//     Term 17 (APS4322-7000)/APS Outputs/Current D 0X1 <-> Data Pointer/DCurrentSetPoints[1]
//     Term 17 (APS4322-7000)/APS Outputs/Current D 0X2 <-> Data Pointer/DCurrentSetPoints[2]
//     Term 17 (APS4322-7000)/APS Outputs/Current D 1X0 <-> Data Pointer/DCurrentSetPoints[6]
//     Term 17 (APS4322-7000)/APS Outputs/Current D 1X1 <-> Data Pointer/DCurrentSetPoints[7]
//     Term 17 (APS4322-7000)/APS Outputs/Current D 1X2 <-> Data Pointer/DCurrentSetPoints[8]
//     Term 17 (APS4322-7000)/APS Outputs/Current D 2X0 <-> Data Pointer/DCurrentSetPoints[12]
//     Term 17 (APS4322-7000)/APS Outputs/Current D 2X1 <-> Data Pointer/DCurrentSetPoints[13]
//     Term 17 (APS4322-7000)/APS Outputs/Current D 2X2 <-> Data Pointer/DCurrentSetPoints[14]
//     Term 17 (APS4322-7000)/APS Outputs/Current D 3X0 <-> Data Pointer/DCurrentSetPoints[18]
//     Term 17 (APS4322-7000)/APS Outputs/Current D 3X1 <-> Data Pointer/DCurrentSetPoints[19]
//     Term 17 (APS4322-7000)/APS Outputs/Current D 3X2 <-> Data Pointer/DCurrentSetPoints[20]
//     Term 17 (APS4322-7000)/APS Outputs/Current D 0Y0 <-> Data Pointer/DCurrentSetPoints[3]
//     Term 17 (APS4322-7000)/APS Outputs/Current D 0Y1 <-> Data Pointer/DCurrentSetPoints[4]
//     Term 17 (APS4322-7000)/APS Outputs/Current D 0Y2 <-> Data Pointer/DCurrentSetPoints[5]
//     Term 17 (APS4322-7000)/APS Outputs/Current D 1Y0 <-> Data Pointer/DCurrentSetPoints[9]
//     Term 17 (APS4322-7000)/APS Outputs/Current D 1Y1 <-> Data Pointer/DCurrentSetPoints[10]
//     Term 17 (APS4322-7000)/APS Outputs/Current D 1Y2 <-> Data Pointer/DCurrentSetPoints[11]
//     Term 17 (APS4322-7000)/APS Outputs/Current D 2Y0 <-> Data Pointer/DCurrentSetPoints[15]
//     Term 17 (APS4322-7000)/APS Outputs/Current D 2Y1 <-> Data Pointer/DCurrentSetPoints[16]
//     Term 17 (APS4322-7000)/APS Outputs/Current D 2Y2 <-> Data Pointer/DCurrentSetPoints[17]
//     Term 17 (APS4322-7000)/APS Outputs/Current D 3Y0 <-> Data Pointer/DCurrentSetPoints[21]
//     Term 17 (APS4322-7000)/APS Outputs/Current D 3Y1 <-> Data Pointer/DCurrentSetPoints[22]
//     Term 17 (APS4322-7000)/APS Outputs/Current D 3Y2 <-> Data Pointer/DCurrentSetPoints[23]
//     Term 17 (APS4322-7000)/APS Outputs/Current Q 0X0 <-> Data Pointer/QCurrentSetPoints[0]
//     Term 17 (APS4322-7000)/APS Outputs/Current Q 0X1 <-> Data Pointer/QCurrentSetPoints[1]
//     Term 17 (APS4322-7000)/APS Outputs/Current Q 0X2 <-> Data Pointer/QCurrentSetPoints[2]
//     Term 17 (APS4322-7000)/APS Outputs/Current Q 1X0 <-> Data Pointer/QCurrentSetPoints[6]
//     Term 17 (APS4322-7000)/APS Outputs/Current Q 1X1 <-> Data Pointer/QCurrentSetPoints[7]
//     Term 17 (APS4322-7000)/APS Outputs/Current Q 1X2 <-> Data Pointer/QCurrentSetPoints[8]
//     Term 17 (APS4322-7000)/APS Outputs/Current Q 2X0 <-> Data Pointer/QCurrentSetPoints[12]
//     Term 17 (APS4322-7000)/APS Outputs/Current Q 2X1 <-> Data Pointer/QCurrentSetPoints[13]
//     Term 17 (APS4322-7000)/APS Outputs/Current Q 2X2 <-> Data Pointer/QCurrentSetPoints[14]
//     Term 17 (APS4322-7000)/APS Outputs/Current Q 3X0 <-> Data Pointer/QCurrentSetPoints[18]
//     Term 17 (APS4322-7000)/APS Outputs/Current Q 3X1 <-> Data Pointer/QCurrentSetPoints[19]
//     Term 17 (APS4322-7000)/APS Outputs/Current Q 3X2 <-> Data Pointer/QCurrentSetPoints[20]
//     Term 17 (APS4322-7000)/APS Outputs/Current Q 0Y0 <-> Data Pointer/QCurrentSetPoints[3]
//     Term 17 (APS4322-7000)/APS Outputs/Current Q 0Y1 <-> Data Pointer/QCurrentSetPoints[4]
//     Term 17 (APS4322-7000)/APS Outputs/Current Q 0Y2 <-> Data Pointer/QCurrentSetPoints[5]
//     Term 17 (APS4322-7000)/APS Outputs/Current Q 1Y0 <-> Data Pointer/QCurrentSetPoints[9]
//     Term 17 (APS4322-7000)/APS Outputs/Current Q 1Y1 <-> Data Pointer/QCurrentSetPoints[10]
//     Term 17 (APS4322-7000)/APS Outputs/Current Q 1Y2 <-> Data Pointer/QCurrentSetPoints[11]
//     Term 17 (APS4322-7000)/APS Outputs/Current Q 2Y0 <-> Data Pointer/QCurrentSetPoints[15]
//     Term 17 (APS4322-7000)/APS Outputs/Current Q 2Y1 <-> Data Pointer/QCurrentSetPoints[16]
//     Term 17 (APS4322-7000)/APS Outputs/Current Q 2Y2 <-> Data Pointer/QCurrentSetPoints[17]
//     Term 17 (APS4322-7000)/APS Outputs/Current Q 3Y0 <-> Data Pointer/QCurrentSetPoints[21]
//     Term 17 (APS4322-7000)/APS Outputs/Current Q 3Y1 <-> Data Pointer/QCurrentSetPoints[22]
//     Term 17 (APS4322-7000)/APS Outputs/Current Q 3Y2 <-> Data Pointer/QCurrentSetPoints[23]
//     Term 17 (APS4322-7000)/APS Outputs/PhiE 0X0 <-> Data Pointer/PhiSetPoints[0]
//     Term 17 (APS4322-7000)/APS Outputs/PhiE 0X1 <-> Data Pointer/PhiSetPoints[1]
//     Term 17 (APS4322-7000)/APS Outputs/PhiE 0X2 <-> Data Pointer/PhiSetPoints[2]
//     Term 17 (APS4322-7000)/APS Outputs/PhiE 1X0 <-> Data Pointer/PhiSetPoints[6]
//     Term 17 (APS4322-7000)/APS Outputs/PhiE 1X1 <-> Data Pointer/PhiSetPoints[7]
//     Term 17 (APS4322-7000)/APS Outputs/PhiE 1X2 <-> Data Pointer/PhiSetPoints[8]
//     Term 17 (APS4322-7000)/APS Outputs/PhiE 2X0 <-> Data Pointer/PhiSetPoints[12]
//     Term 17 (APS4322-7000)/APS Outputs/PhiE 2X1 <-> Data Pointer/PhiSetPoints[13]
//     Term 17 (APS4322-7000)/APS Outputs/PhiE 2X2 <-> Data Pointer/PhiSetPoints[14]
//     Term 17 (APS4322-7000)/APS Outputs/PhiE 3X0 <-> Data Pointer/PhiSetPoints[18]
//     Term 17 (APS4322-7000)/APS Outputs/PhiE 3X1 <-> Data Pointer/PhiSetPoints[19]
//     Term 17 (APS4322-7000)/APS Outputs/PhiE 3X2 <-> Data Pointer/PhiSetPoints[20]
//     Term 17 (APS4322-7000)/APS Outputs/PhiE 0Y0 <-> Data Pointer/PhiSetPoints[3]
//     Term 17 (APS4322-7000)/APS Outputs/PhiE 0Y1 <-> Data Pointer/PhiSetPoints[4]
//     Term 17 (APS4322-7000)/APS Outputs/PhiE 0Y2 <-> Data Pointer/PhiSetPoints[5]
//     Term 17 (APS4322-7000)/APS Outputs/PhiE 1Y0 <-> Data Pointer/PhiSetPoints[9]
//     Term 17 (APS4322-7000)/APS Outputs/PhiE 1Y1 <-> Data Pointer/PhiSetPoints[10]
//     Term 17 (APS4322-7000)/APS Outputs/PhiE 1Y2 <-> Data Pointer/PhiSetPoints[11]
//     Term 17 (APS4322-7000)/APS Outputs/PhiE 2Y0 <-> Data Pointer/PhiSetPoints[15]
//     Term 17 (APS4322-7000)/APS Outputs/PhiE 2Y1 <-> Data Pointer/PhiSetPoints[16]
//     Term 17 (APS4322-7000)/APS Outputs/PhiE 2Y2 <-> Data Pointer/PhiSetPoints[17]
//     Term 17 (APS4322-7000)/APS Outputs/PhiE 3Y0 <-> Data Pointer/PhiSetPoints[21]
//     Term 17 (APS4322-7000)/APS Outputs/PhiE 3Y1 <-> Data Pointer/PhiSetPoints[22]
//     Term 17 (APS4322-7000)/APS Outputs/PhiE 3Y2 <-> Data Pointer/PhiSetPoints[23]
//     Term 17 (APS4322-7000)/Term 18 (APS4322-5000)/FB Inputs/A{0..8 step 2} X-Field <-> Data Pointer/HallSensorFieldsXYZ[{0..12 step 3}]  (5 links)
//     Term 17 (APS4322-7000)/Term 18 (APS4322-5000)/FB Inputs/A{0..8 step 2} Y-Field <-> Data Pointer/HallSensorFieldsXYZ[{1..13 step 3}]  (5 links)
//     Term 17 (APS4322-7000)/Term 18 (APS4322-5000)/FB Inputs/A{0..8 step 2} Z-Field <-> Data Pointer/HallSensorFieldsXYZ[{2..14 step 3}]  (5 links)
//     Term 17 (APS4322-7000)/Term 18 (APS4322-5000)/FB Inputs/B{1..9 step 2} X-Field <-> Data Pointer/HallSensorFieldsXYZ[{15..27 step 3}]  (5 links)
//     Term 17 (APS4322-7000)/Term 18 (APS4322-5000)/FB Inputs/B{1..9 step 2} Y-Field <-> Data Pointer/HallSensorFieldsXYZ[{16..28 step 3}]  (5 links)
//     Term 17 (APS4322-7000)/Term 18 (APS4322-5000)/FB Inputs/B{1..9 step 2} Z-Field <-> Data Pointer/HallSensorFieldsXYZ[{17..29 step 3}]  (5 links)
//     Term 17 (APS4322-7000)/Term 18 (APS4322-5000)/FB Inputs/C{0..8 step 2} X-Field <-> Data Pointer/HallSensorFieldsXYZ[{30..42 step 3}]  (5 links)
//     Term 17 (APS4322-7000)/Term 18 (APS4322-5000)/FB Inputs/C{0..8 step 2} Y-Field <-> Data Pointer/HallSensorFieldsXYZ[{31..43 step 3}]  (5 links)
//     Term 17 (APS4322-7000)/Term 18 (APS4322-5000)/FB Inputs/C{0..8 step 2} Z-Field <-> Data Pointer/HallSensorFieldsXYZ[{32..44 step 3}]  (5 links)
//     Term 17 (APS4322-7000)/Term 18 (APS4322-5000)/FB Inputs/D{1..9 step 2} X-Field <-> Data Pointer/HallSensorFieldsXYZ[{45..57 step 3}]  (5 links)
//     Term 17 (APS4322-7000)/Term 18 (APS4322-5000)/FB Inputs/D{1..9 step 2} Y-Field <-> Data Pointer/HallSensorFieldsXYZ[{46..58 step 3}]  (5 links)
//     Term 17 (APS4322-7000)/Term 18 (APS4322-5000)/FB Inputs/D{1..9 step 2} Z-Field <-> Data Pointer/HallSensorFieldsXYZ[{47..59 step 3}]  (5 links)
//     Term 17 (APS4322-7000)/Term 18 (APS4322-5000)/FB Inputs/E{0..8 step 2} X-Field <-> Data Pointer/HallSensorFieldsXYZ[{60..72 step 3}]  (5 links)
//     Term 17 (APS4322-7000)/Term 18 (APS4322-5000)/FB Inputs/E{0..8 step 2} Y-Field <-> Data Pointer/HallSensorFieldsXYZ[{61..73 step 3}]  (5 links)
//     Term 17 (APS4322-7000)/Term 18 (APS4322-5000)/FB Inputs/E{0..8 step 2} Z-Field <-> Data Pointer/HallSensorFieldsXYZ[{62..74 step 3}]  (5 links)
//     Term 17 (APS4322-7000)/Term 18 (APS4322-5000)/FB Inputs/F{1..9 step 2} X-Field <-> Data Pointer/HallSensorFieldsXYZ[{75..87 step 3}]  (5 links)
//     Term 17 (APS4322-7000)/Term 18 (APS4322-5000)/FB Inputs/F{1..9 step 2} Y-Field <-> Data Pointer/HallSensorFieldsXYZ[{76..88 step 3}]  (5 links)
//     Term 17 (APS4322-7000)/Term 18 (APS4322-5000)/FB Inputs/F{1..9 step 2} Z-Field <-> Data Pointer/HallSensorFieldsXYZ[{77..89 step 3}]  (5 links)
//     Term 17 (APS4322-7000)/Term 18 (APS4322-5000)/FB Inputs/G{0..8 step 2} X-Field <-> Data Pointer/HallSensorFieldsXYZ[{90..102 step 3}]  (5 links)
//     Term 17 (APS4322-7000)/Term 18 (APS4322-5000)/FB Inputs/G{0..8 step 2} Y-Field <-> Data Pointer/HallSensorFieldsXYZ[{91..103 step 3}]  (5 links)
//     Term 17 (APS4322-7000)/Term 18 (APS4322-5000)/FB Inputs/G{0..8 step 2} Z-Field <-> Data Pointer/HallSensorFieldsXYZ[{92..104 step 3}]  (5 links)
//     Term 17 (APS4322-7000)/Term 18 (APS4322-5000)/FB Inputs/H{1..9 step 2} X-Field <-> Data Pointer/HallSensorFieldsXYZ[{105..117 step 3}]  (5 links)
//     Term 17 (APS4322-7000)/Term 18 (APS4322-5000)/FB Inputs/H{1..9 step 2} Y-Field <-> Data Pointer/HallSensorFieldsXYZ[{106..118 step 3}]  (5 links)
//     Term 17 (APS4322-7000)/Term 18 (APS4322-5000)/FB Inputs/H{1..9 step 2} Z-Field <-> Data Pointer/HallSensorFieldsXYZ[{107..119 step 3}]  (5 links)
//     Term 17 (APS4322-7000)/Term 18 (APS4322-5000)/FB Inputs/I{0..8 step 2} X-Field <-> Data Pointer/HallSensorFieldsXYZ[{120..132 step 3}]  (5 links)
//     Term 17 (APS4322-7000)/Term 18 (APS4322-5000)/FB Inputs/I{0..8 step 2} Y-Field <-> Data Pointer/HallSensorFieldsXYZ[{121..133 step 3}]  (5 links)
//     Term 17 (APS4322-7000)/Term 18 (APS4322-5000)/FB Inputs/I{0..8 step 2} Z-Field <-> Data Pointer/HallSensorFieldsXYZ[{122..134 step 3}]  (5 links)
//     Term 17 (APS4322-7000)/Term 18 (APS4322-5000)/FB Inputs/J{1..9 step 2} X-Field <-> Data Pointer/HallSensorFieldsXYZ[{135..147 step 3}]  (5 links)
//     Term 17 (APS4322-7000)/Term 18 (APS4322-5000)/FB Inputs/J{1..9 step 2} Y-Field <-> Data Pointer/HallSensorFieldsXYZ[{136..148 step 3}]  (5 links)
//     Term 17 (APS4322-7000)/Term 18 (APS4322-5000)/FB Inputs/J{1..9 step 2} Z-Field <-> Data Pointer/HallSensorFieldsXYZ[{137..149 step 3}]  (5 links)
//     Term 17 (APS4322-7000)/Term 18 (APS4322-5000)/FB Inputs/Status <-> Data Pointer/FeedbackStatus
//   Device 2 (EtherCAT) <-> TcCOM Objects/XPlanar/Part1/Tile4
//     Term 19 (APS4322-7000)/APS Comm Inputs/CommStatusWord <-> Data Pointer/MoverCommStatusWord
//     Term 19 (APS4322-7000)/APS Comm Inputs/Data {1..4} <-> Data Pointer/MoverCommDataIn[{0..3}]  (4 links)
//     Term 19 (APS4322-7000)/APS Comm Outputs/CommControlWord <-> Data Pointer/MoverCommControlWord
//     Term 19 (APS4322-7000)/APS Comm Outputs/Data 1 <-> Data Pointer/MoverCommDataOut
//     Term 19 (APS4322-7000)/APS Diagdata/DC Link Voltage <-> Data Pointer/DcLinkVoltage
//     Term 19 (APS4322-7000)/APS Diagdata/Power supply current <-> Data Pointer/PowerSupplyCurrent
//     Term 19 (APS4322-7000)/APS Inputs/StatusWord <-> Data Pointer/PowerUnitStatusWord
//     Term 19 (APS4322-7000)/APS Outputs/ControlWord <-> Data Pointer/PowerUnitControlWord
//     Term 19 (APS4322-7000)/APS Outputs/Current D 0X0 <-> Data Pointer/DCurrentSetPoints[0]
//     Term 19 (APS4322-7000)/APS Outputs/Current D 0X1 <-> Data Pointer/DCurrentSetPoints[1]
//     Term 19 (APS4322-7000)/APS Outputs/Current D 0X2 <-> Data Pointer/DCurrentSetPoints[2]
//     Term 19 (APS4322-7000)/APS Outputs/Current D 1X0 <-> Data Pointer/DCurrentSetPoints[6]
//     Term 19 (APS4322-7000)/APS Outputs/Current D 1X1 <-> Data Pointer/DCurrentSetPoints[7]
//     Term 19 (APS4322-7000)/APS Outputs/Current D 1X2 <-> Data Pointer/DCurrentSetPoints[8]
//     Term 19 (APS4322-7000)/APS Outputs/Current D 2X0 <-> Data Pointer/DCurrentSetPoints[12]
//     Term 19 (APS4322-7000)/APS Outputs/Current D 2X1 <-> Data Pointer/DCurrentSetPoints[13]
//     Term 19 (APS4322-7000)/APS Outputs/Current D 2X2 <-> Data Pointer/DCurrentSetPoints[14]
//     Term 19 (APS4322-7000)/APS Outputs/Current D 3X0 <-> Data Pointer/DCurrentSetPoints[18]
//     Term 19 (APS4322-7000)/APS Outputs/Current D 3X1 <-> Data Pointer/DCurrentSetPoints[19]
//     Term 19 (APS4322-7000)/APS Outputs/Current D 3X2 <-> Data Pointer/DCurrentSetPoints[20]
//     Term 19 (APS4322-7000)/APS Outputs/Current D 0Y0 <-> Data Pointer/DCurrentSetPoints[3]
//     Term 19 (APS4322-7000)/APS Outputs/Current D 0Y1 <-> Data Pointer/DCurrentSetPoints[4]
//     Term 19 (APS4322-7000)/APS Outputs/Current D 0Y2 <-> Data Pointer/DCurrentSetPoints[5]
//     Term 19 (APS4322-7000)/APS Outputs/Current D 1Y0 <-> Data Pointer/DCurrentSetPoints[9]
//     Term 19 (APS4322-7000)/APS Outputs/Current D 1Y1 <-> Data Pointer/DCurrentSetPoints[10]
//     Term 19 (APS4322-7000)/APS Outputs/Current D 1Y2 <-> Data Pointer/DCurrentSetPoints[11]
//     Term 19 (APS4322-7000)/APS Outputs/Current D 2Y0 <-> Data Pointer/DCurrentSetPoints[15]
//     Term 19 (APS4322-7000)/APS Outputs/Current D 2Y1 <-> Data Pointer/DCurrentSetPoints[16]
//     Term 19 (APS4322-7000)/APS Outputs/Current D 2Y2 <-> Data Pointer/DCurrentSetPoints[17]
//     Term 19 (APS4322-7000)/APS Outputs/Current D 3Y0 <-> Data Pointer/DCurrentSetPoints[21]
//     Term 19 (APS4322-7000)/APS Outputs/Current D 3Y1 <-> Data Pointer/DCurrentSetPoints[22]
//     Term 19 (APS4322-7000)/APS Outputs/Current D 3Y2 <-> Data Pointer/DCurrentSetPoints[23]
//     Term 19 (APS4322-7000)/APS Outputs/Current Q 0X0 <-> Data Pointer/QCurrentSetPoints[0]
//     Term 19 (APS4322-7000)/APS Outputs/Current Q 0X1 <-> Data Pointer/QCurrentSetPoints[1]
//     Term 19 (APS4322-7000)/APS Outputs/Current Q 0X2 <-> Data Pointer/QCurrentSetPoints[2]
//     Term 19 (APS4322-7000)/APS Outputs/Current Q 1X0 <-> Data Pointer/QCurrentSetPoints[6]
//     Term 19 (APS4322-7000)/APS Outputs/Current Q 1X1 <-> Data Pointer/QCurrentSetPoints[7]
//     Term 19 (APS4322-7000)/APS Outputs/Current Q 1X2 <-> Data Pointer/QCurrentSetPoints[8]
//     Term 19 (APS4322-7000)/APS Outputs/Current Q 2X0 <-> Data Pointer/QCurrentSetPoints[12]
//     Term 19 (APS4322-7000)/APS Outputs/Current Q 2X1 <-> Data Pointer/QCurrentSetPoints[13]
//     Term 19 (APS4322-7000)/APS Outputs/Current Q 2X2 <-> Data Pointer/QCurrentSetPoints[14]
//     Term 19 (APS4322-7000)/APS Outputs/Current Q 3X0 <-> Data Pointer/QCurrentSetPoints[18]
//     Term 19 (APS4322-7000)/APS Outputs/Current Q 3X1 <-> Data Pointer/QCurrentSetPoints[19]
//     Term 19 (APS4322-7000)/APS Outputs/Current Q 3X2 <-> Data Pointer/QCurrentSetPoints[20]
//     Term 19 (APS4322-7000)/APS Outputs/Current Q 0Y0 <-> Data Pointer/QCurrentSetPoints[3]
//     Term 19 (APS4322-7000)/APS Outputs/Current Q 0Y1 <-> Data Pointer/QCurrentSetPoints[4]
//     Term 19 (APS4322-7000)/APS Outputs/Current Q 0Y2 <-> Data Pointer/QCurrentSetPoints[5]
//     Term 19 (APS4322-7000)/APS Outputs/Current Q 1Y0 <-> Data Pointer/QCurrentSetPoints[9]
//     Term 19 (APS4322-7000)/APS Outputs/Current Q 1Y1 <-> Data Pointer/QCurrentSetPoints[10]
//     Term 19 (APS4322-7000)/APS Outputs/Current Q 1Y2 <-> Data Pointer/QCurrentSetPoints[11]
//     Term 19 (APS4322-7000)/APS Outputs/Current Q 2Y0 <-> Data Pointer/QCurrentSetPoints[15]
//     Term 19 (APS4322-7000)/APS Outputs/Current Q 2Y1 <-> Data Pointer/QCurrentSetPoints[16]
//     Term 19 (APS4322-7000)/APS Outputs/Current Q 2Y2 <-> Data Pointer/QCurrentSetPoints[17]
//     Term 19 (APS4322-7000)/APS Outputs/Current Q 3Y0 <-> Data Pointer/QCurrentSetPoints[21]
//     Term 19 (APS4322-7000)/APS Outputs/Current Q 3Y1 <-> Data Pointer/QCurrentSetPoints[22]
//     Term 19 (APS4322-7000)/APS Outputs/Current Q 3Y2 <-> Data Pointer/QCurrentSetPoints[23]
//     Term 19 (APS4322-7000)/APS Outputs/PhiE 0X0 <-> Data Pointer/PhiSetPoints[0]
//     Term 19 (APS4322-7000)/APS Outputs/PhiE 0X1 <-> Data Pointer/PhiSetPoints[1]
//     Term 19 (APS4322-7000)/APS Outputs/PhiE 0X2 <-> Data Pointer/PhiSetPoints[2]
//     Term 19 (APS4322-7000)/APS Outputs/PhiE 1X0 <-> Data Pointer/PhiSetPoints[6]
//     Term 19 (APS4322-7000)/APS Outputs/PhiE 1X1 <-> Data Pointer/PhiSetPoints[7]
//     Term 19 (APS4322-7000)/APS Outputs/PhiE 1X2 <-> Data Pointer/PhiSetPoints[8]
//     Term 19 (APS4322-7000)/APS Outputs/PhiE 2X0 <-> Data Pointer/PhiSetPoints[12]
//     Term 19 (APS4322-7000)/APS Outputs/PhiE 2X1 <-> Data Pointer/PhiSetPoints[13]
//     Term 19 (APS4322-7000)/APS Outputs/PhiE 2X2 <-> Data Pointer/PhiSetPoints[14]
//     Term 19 (APS4322-7000)/APS Outputs/PhiE 3X0 <-> Data Pointer/PhiSetPoints[18]
//     Term 19 (APS4322-7000)/APS Outputs/PhiE 3X1 <-> Data Pointer/PhiSetPoints[19]
//     Term 19 (APS4322-7000)/APS Outputs/PhiE 3X2 <-> Data Pointer/PhiSetPoints[20]
//     Term 19 (APS4322-7000)/APS Outputs/PhiE 0Y0 <-> Data Pointer/PhiSetPoints[3]
//     Term 19 (APS4322-7000)/APS Outputs/PhiE 0Y1 <-> Data Pointer/PhiSetPoints[4]
//     Term 19 (APS4322-7000)/APS Outputs/PhiE 0Y2 <-> Data Pointer/PhiSetPoints[5]
//     Term 19 (APS4322-7000)/APS Outputs/PhiE 1Y0 <-> Data Pointer/PhiSetPoints[9]
//     Term 19 (APS4322-7000)/APS Outputs/PhiE 1Y1 <-> Data Pointer/PhiSetPoints[10]
//     Term 19 (APS4322-7000)/APS Outputs/PhiE 1Y2 <-> Data Pointer/PhiSetPoints[11]
//     Term 19 (APS4322-7000)/APS Outputs/PhiE 2Y0 <-> Data Pointer/PhiSetPoints[15]
//     Term 19 (APS4322-7000)/APS Outputs/PhiE 2Y1 <-> Data Pointer/PhiSetPoints[16]
//     Term 19 (APS4322-7000)/APS Outputs/PhiE 2Y2 <-> Data Pointer/PhiSetPoints[17]
//     Term 19 (APS4322-7000)/APS Outputs/PhiE 3Y0 <-> Data Pointer/PhiSetPoints[21]
//     Term 19 (APS4322-7000)/APS Outputs/PhiE 3Y1 <-> Data Pointer/PhiSetPoints[22]
//     Term 19 (APS4322-7000)/APS Outputs/PhiE 3Y2 <-> Data Pointer/PhiSetPoints[23]
//     Term 19 (APS4322-7000)/Term 20 (APS4322-5000)/FB Inputs/A{0..8 step 2} X-Field <-> Data Pointer/HallSensorFieldsXYZ[{0..12 step 3}]  (5 links)
//     Term 19 (APS4322-7000)/Term 20 (APS4322-5000)/FB Inputs/A{0..8 step 2} Y-Field <-> Data Pointer/HallSensorFieldsXYZ[{1..13 step 3}]  (5 links)
//     Term 19 (APS4322-7000)/Term 20 (APS4322-5000)/FB Inputs/A{0..8 step 2} Z-Field <-> Data Pointer/HallSensorFieldsXYZ[{2..14 step 3}]  (5 links)
//     Term 19 (APS4322-7000)/Term 20 (APS4322-5000)/FB Inputs/B{1..9 step 2} X-Field <-> Data Pointer/HallSensorFieldsXYZ[{15..27 step 3}]  (5 links)
//     Term 19 (APS4322-7000)/Term 20 (APS4322-5000)/FB Inputs/B{1..9 step 2} Y-Field <-> Data Pointer/HallSensorFieldsXYZ[{16..28 step 3}]  (5 links)
//     Term 19 (APS4322-7000)/Term 20 (APS4322-5000)/FB Inputs/B{1..9 step 2} Z-Field <-> Data Pointer/HallSensorFieldsXYZ[{17..29 step 3}]  (5 links)
//     Term 19 (APS4322-7000)/Term 20 (APS4322-5000)/FB Inputs/C{0..8 step 2} X-Field <-> Data Pointer/HallSensorFieldsXYZ[{30..42 step 3}]  (5 links)
//     Term 19 (APS4322-7000)/Term 20 (APS4322-5000)/FB Inputs/C{0..8 step 2} Y-Field <-> Data Pointer/HallSensorFieldsXYZ[{31..43 step 3}]  (5 links)
//     Term 19 (APS4322-7000)/Term 20 (APS4322-5000)/FB Inputs/C{0..8 step 2} Z-Field <-> Data Pointer/HallSensorFieldsXYZ[{32..44 step 3}]  (5 links)
//     Term 19 (APS4322-7000)/Term 20 (APS4322-5000)/FB Inputs/D{1..9 step 2} X-Field <-> Data Pointer/HallSensorFieldsXYZ[{45..57 step 3}]  (5 links)
//     Term 19 (APS4322-7000)/Term 20 (APS4322-5000)/FB Inputs/D{1..9 step 2} Y-Field <-> Data Pointer/HallSensorFieldsXYZ[{46..58 step 3}]  (5 links)
//     Term 19 (APS4322-7000)/Term 20 (APS4322-5000)/FB Inputs/D{1..9 step 2} Z-Field <-> Data Pointer/HallSensorFieldsXYZ[{47..59 step 3}]  (5 links)
//     Term 19 (APS4322-7000)/Term 20 (APS4322-5000)/FB Inputs/E{0..8 step 2} X-Field <-> Data Pointer/HallSensorFieldsXYZ[{60..72 step 3}]  (5 links)
//     Term 19 (APS4322-7000)/Term 20 (APS4322-5000)/FB Inputs/E{0..8 step 2} Y-Field <-> Data Pointer/HallSensorFieldsXYZ[{61..73 step 3}]  (5 links)
//     Term 19 (APS4322-7000)/Term 20 (APS4322-5000)/FB Inputs/E{0..8 step 2} Z-Field <-> Data Pointer/HallSensorFieldsXYZ[{62..74 step 3}]  (5 links)
//     Term 19 (APS4322-7000)/Term 20 (APS4322-5000)/FB Inputs/F{1..9 step 2} X-Field <-> Data Pointer/HallSensorFieldsXYZ[{75..87 step 3}]  (5 links)
//     Term 19 (APS4322-7000)/Term 20 (APS4322-5000)/FB Inputs/F{1..9 step 2} Y-Field <-> Data Pointer/HallSensorFieldsXYZ[{76..88 step 3}]  (5 links)
//     Term 19 (APS4322-7000)/Term 20 (APS4322-5000)/FB Inputs/F{1..9 step 2} Z-Field <-> Data Pointer/HallSensorFieldsXYZ[{77..89 step 3}]  (5 links)
//     Term 19 (APS4322-7000)/Term 20 (APS4322-5000)/FB Inputs/G{0..8 step 2} X-Field <-> Data Pointer/HallSensorFieldsXYZ[{90..102 step 3}]  (5 links)
//     Term 19 (APS4322-7000)/Term 20 (APS4322-5000)/FB Inputs/G{0..8 step 2} Y-Field <-> Data Pointer/HallSensorFieldsXYZ[{91..103 step 3}]  (5 links)
//     Term 19 (APS4322-7000)/Term 20 (APS4322-5000)/FB Inputs/G{0..8 step 2} Z-Field <-> Data Pointer/HallSensorFieldsXYZ[{92..104 step 3}]  (5 links)
//     Term 19 (APS4322-7000)/Term 20 (APS4322-5000)/FB Inputs/H{1..9 step 2} X-Field <-> Data Pointer/HallSensorFieldsXYZ[{105..117 step 3}]  (5 links)
//     Term 19 (APS4322-7000)/Term 20 (APS4322-5000)/FB Inputs/H{1..9 step 2} Y-Field <-> Data Pointer/HallSensorFieldsXYZ[{106..118 step 3}]  (5 links)
//     Term 19 (APS4322-7000)/Term 20 (APS4322-5000)/FB Inputs/H{1..9 step 2} Z-Field <-> Data Pointer/HallSensorFieldsXYZ[{107..119 step 3}]  (5 links)
//     Term 19 (APS4322-7000)/Term 20 (APS4322-5000)/FB Inputs/I{0..8 step 2} X-Field <-> Data Pointer/HallSensorFieldsXYZ[{120..132 step 3}]  (5 links)
//     Term 19 (APS4322-7000)/Term 20 (APS4322-5000)/FB Inputs/I{0..8 step 2} Y-Field <-> Data Pointer/HallSensorFieldsXYZ[{121..133 step 3}]  (5 links)
//     Term 19 (APS4322-7000)/Term 20 (APS4322-5000)/FB Inputs/I{0..8 step 2} Z-Field <-> Data Pointer/HallSensorFieldsXYZ[{122..134 step 3}]  (5 links)
//     Term 19 (APS4322-7000)/Term 20 (APS4322-5000)/FB Inputs/J{1..9 step 2} X-Field <-> Data Pointer/HallSensorFieldsXYZ[{135..147 step 3}]  (5 links)
//     Term 19 (APS4322-7000)/Term 20 (APS4322-5000)/FB Inputs/J{1..9 step 2} Y-Field <-> Data Pointer/HallSensorFieldsXYZ[{136..148 step 3}]  (5 links)
//     Term 19 (APS4322-7000)/Term 20 (APS4322-5000)/FB Inputs/J{1..9 step 2} Z-Field <-> Data Pointer/HallSensorFieldsXYZ[{137..149 step 3}]  (5 links)
//     Term 19 (APS4322-7000)/Term 20 (APS4322-5000)/FB Inputs/Status <-> Data Pointer/FeedbackStatus
//   Device 2 (EtherCAT) <-> TcCOM Objects/XPlanar/Part1/Tile7
//     Term 21 (APS4322-7000)/APS Comm Inputs/CommStatusWord <-> Data Pointer/MoverCommStatusWord
//     Term 21 (APS4322-7000)/APS Comm Inputs/Data {1..4} <-> Data Pointer/MoverCommDataIn[{0..3}]  (4 links)
//     Term 21 (APS4322-7000)/APS Comm Outputs/CommControlWord <-> Data Pointer/MoverCommControlWord
//     Term 21 (APS4322-7000)/APS Comm Outputs/Data 1 <-> Data Pointer/MoverCommDataOut
//     Term 21 (APS4322-7000)/APS Diagdata/DC Link Voltage <-> Data Pointer/DcLinkVoltage
//     Term 21 (APS4322-7000)/APS Diagdata/Power supply current <-> Data Pointer/PowerSupplyCurrent
//     Term 21 (APS4322-7000)/APS Inputs/StatusWord <-> Data Pointer/PowerUnitStatusWord
//     Term 21 (APS4322-7000)/APS Outputs/ControlWord <-> Data Pointer/PowerUnitControlWord
//     Term 21 (APS4322-7000)/APS Outputs/Current D 0X0 <-> Data Pointer/DCurrentSetPoints[0]
//     Term 21 (APS4322-7000)/APS Outputs/Current D 0X1 <-> Data Pointer/DCurrentSetPoints[1]
//     Term 21 (APS4322-7000)/APS Outputs/Current D 0X2 <-> Data Pointer/DCurrentSetPoints[2]
//     Term 21 (APS4322-7000)/APS Outputs/Current D 1X0 <-> Data Pointer/DCurrentSetPoints[6]
//     Term 21 (APS4322-7000)/APS Outputs/Current D 1X1 <-> Data Pointer/DCurrentSetPoints[7]
//     Term 21 (APS4322-7000)/APS Outputs/Current D 1X2 <-> Data Pointer/DCurrentSetPoints[8]
//     Term 21 (APS4322-7000)/APS Outputs/Current D 2X0 <-> Data Pointer/DCurrentSetPoints[12]
//     Term 21 (APS4322-7000)/APS Outputs/Current D 2X1 <-> Data Pointer/DCurrentSetPoints[13]
//     Term 21 (APS4322-7000)/APS Outputs/Current D 2X2 <-> Data Pointer/DCurrentSetPoints[14]
//     Term 21 (APS4322-7000)/APS Outputs/Current D 3X0 <-> Data Pointer/DCurrentSetPoints[18]
//     Term 21 (APS4322-7000)/APS Outputs/Current D 3X1 <-> Data Pointer/DCurrentSetPoints[19]
//     Term 21 (APS4322-7000)/APS Outputs/Current D 3X2 <-> Data Pointer/DCurrentSetPoints[20]
//     Term 21 (APS4322-7000)/APS Outputs/Current D 0Y0 <-> Data Pointer/DCurrentSetPoints[3]
//     Term 21 (APS4322-7000)/APS Outputs/Current D 0Y1 <-> Data Pointer/DCurrentSetPoints[4]
//     Term 21 (APS4322-7000)/APS Outputs/Current D 0Y2 <-> Data Pointer/DCurrentSetPoints[5]
//     Term 21 (APS4322-7000)/APS Outputs/Current D 1Y0 <-> Data Pointer/DCurrentSetPoints[9]
//     Term 21 (APS4322-7000)/APS Outputs/Current D 1Y1 <-> Data Pointer/DCurrentSetPoints[10]
//     Term 21 (APS4322-7000)/APS Outputs/Current D 1Y2 <-> Data Pointer/DCurrentSetPoints[11]
//     Term 21 (APS4322-7000)/APS Outputs/Current D 2Y0 <-> Data Pointer/DCurrentSetPoints[15]
//     Term 21 (APS4322-7000)/APS Outputs/Current D 2Y1 <-> Data Pointer/DCurrentSetPoints[16]
//     Term 21 (APS4322-7000)/APS Outputs/Current D 2Y2 <-> Data Pointer/DCurrentSetPoints[17]
//     Term 21 (APS4322-7000)/APS Outputs/Current D 3Y0 <-> Data Pointer/DCurrentSetPoints[21]
//     Term 21 (APS4322-7000)/APS Outputs/Current D 3Y1 <-> Data Pointer/DCurrentSetPoints[22]
//     Term 21 (APS4322-7000)/APS Outputs/Current D 3Y2 <-> Data Pointer/DCurrentSetPoints[23]
//     Term 21 (APS4322-7000)/APS Outputs/Current Q 0X0 <-> Data Pointer/QCurrentSetPoints[0]
//     Term 21 (APS4322-7000)/APS Outputs/Current Q 0X1 <-> Data Pointer/QCurrentSetPoints[1]
//     Term 21 (APS4322-7000)/APS Outputs/Current Q 0X2 <-> Data Pointer/QCurrentSetPoints[2]
//     Term 21 (APS4322-7000)/APS Outputs/Current Q 1X0 <-> Data Pointer/QCurrentSetPoints[6]
//     Term 21 (APS4322-7000)/APS Outputs/Current Q 1X1 <-> Data Pointer/QCurrentSetPoints[7]
//     Term 21 (APS4322-7000)/APS Outputs/Current Q 1X2 <-> Data Pointer/QCurrentSetPoints[8]
//     Term 21 (APS4322-7000)/APS Outputs/Current Q 2X0 <-> Data Pointer/QCurrentSetPoints[12]
//     Term 21 (APS4322-7000)/APS Outputs/Current Q 2X1 <-> Data Pointer/QCurrentSetPoints[13]
//     Term 21 (APS4322-7000)/APS Outputs/Current Q 2X2 <-> Data Pointer/QCurrentSetPoints[14]
//     Term 21 (APS4322-7000)/APS Outputs/Current Q 3X0 <-> Data Pointer/QCurrentSetPoints[18]
//     Term 21 (APS4322-7000)/APS Outputs/Current Q 3X1 <-> Data Pointer/QCurrentSetPoints[19]
//     Term 21 (APS4322-7000)/APS Outputs/Current Q 3X2 <-> Data Pointer/QCurrentSetPoints[20]
//     Term 21 (APS4322-7000)/APS Outputs/Current Q 0Y0 <-> Data Pointer/QCurrentSetPoints[3]
//     Term 21 (APS4322-7000)/APS Outputs/Current Q 0Y1 <-> Data Pointer/QCurrentSetPoints[4]
//     Term 21 (APS4322-7000)/APS Outputs/Current Q 0Y2 <-> Data Pointer/QCurrentSetPoints[5]
//     Term 21 (APS4322-7000)/APS Outputs/Current Q 1Y0 <-> Data Pointer/QCurrentSetPoints[9]
//     Term 21 (APS4322-7000)/APS Outputs/Current Q 1Y1 <-> Data Pointer/QCurrentSetPoints[10]
//     Term 21 (APS4322-7000)/APS Outputs/Current Q 1Y2 <-> Data Pointer/QCurrentSetPoints[11]
//     Term 21 (APS4322-7000)/APS Outputs/Current Q 2Y0 <-> Data Pointer/QCurrentSetPoints[15]
//     Term 21 (APS4322-7000)/APS Outputs/Current Q 2Y1 <-> Data Pointer/QCurrentSetPoints[16]
//     Term 21 (APS4322-7000)/APS Outputs/Current Q 2Y2 <-> Data Pointer/QCurrentSetPoints[17]
//     Term 21 (APS4322-7000)/APS Outputs/Current Q 3Y0 <-> Data Pointer/QCurrentSetPoints[21]
//     Term 21 (APS4322-7000)/APS Outputs/Current Q 3Y1 <-> Data Pointer/QCurrentSetPoints[22]
//     Term 21 (APS4322-7000)/APS Outputs/Current Q 3Y2 <-> Data Pointer/QCurrentSetPoints[23]
//     Term 21 (APS4322-7000)/APS Outputs/PhiE 0X0 <-> Data Pointer/PhiSetPoints[0]
//     Term 21 (APS4322-7000)/APS Outputs/PhiE 0X1 <-> Data Pointer/PhiSetPoints[1]
//     Term 21 (APS4322-7000)/APS Outputs/PhiE 0X2 <-> Data Pointer/PhiSetPoints[2]
//     Term 21 (APS4322-7000)/APS Outputs/PhiE 1X0 <-> Data Pointer/PhiSetPoints[6]
//     Term 21 (APS4322-7000)/APS Outputs/PhiE 1X1 <-> Data Pointer/PhiSetPoints[7]
//     Term 21 (APS4322-7000)/APS Outputs/PhiE 1X2 <-> Data Pointer/PhiSetPoints[8]
//     Term 21 (APS4322-7000)/APS Outputs/PhiE 2X0 <-> Data Pointer/PhiSetPoints[12]
//     Term 21 (APS4322-7000)/APS Outputs/PhiE 2X1 <-> Data Pointer/PhiSetPoints[13]
//     Term 21 (APS4322-7000)/APS Outputs/PhiE 2X2 <-> Data Pointer/PhiSetPoints[14]
//     Term 21 (APS4322-7000)/APS Outputs/PhiE 3X0 <-> Data Pointer/PhiSetPoints[18]
//     Term 21 (APS4322-7000)/APS Outputs/PhiE 3X1 <-> Data Pointer/PhiSetPoints[19]
//     Term 21 (APS4322-7000)/APS Outputs/PhiE 3X2 <-> Data Pointer/PhiSetPoints[20]
//     Term 21 (APS4322-7000)/APS Outputs/PhiE 0Y0 <-> Data Pointer/PhiSetPoints[3]
//     Term 21 (APS4322-7000)/APS Outputs/PhiE 0Y1 <-> Data Pointer/PhiSetPoints[4]
//     Term 21 (APS4322-7000)/APS Outputs/PhiE 0Y2 <-> Data Pointer/PhiSetPoints[5]
//     Term 21 (APS4322-7000)/APS Outputs/PhiE 1Y0 <-> Data Pointer/PhiSetPoints[9]
//     Term 21 (APS4322-7000)/APS Outputs/PhiE 1Y1 <-> Data Pointer/PhiSetPoints[10]
//     Term 21 (APS4322-7000)/APS Outputs/PhiE 1Y2 <-> Data Pointer/PhiSetPoints[11]
//     Term 21 (APS4322-7000)/APS Outputs/PhiE 2Y0 <-> Data Pointer/PhiSetPoints[15]
//     Term 21 (APS4322-7000)/APS Outputs/PhiE 2Y1 <-> Data Pointer/PhiSetPoints[16]
//     Term 21 (APS4322-7000)/APS Outputs/PhiE 2Y2 <-> Data Pointer/PhiSetPoints[17]
//     Term 21 (APS4322-7000)/APS Outputs/PhiE 3Y0 <-> Data Pointer/PhiSetPoints[21]
//     Term 21 (APS4322-7000)/APS Outputs/PhiE 3Y1 <-> Data Pointer/PhiSetPoints[22]
//     Term 21 (APS4322-7000)/APS Outputs/PhiE 3Y2 <-> Data Pointer/PhiSetPoints[23]
//     Term 21 (APS4322-7000)/Term 22 (APS4322-5000)/FB Inputs/A{0..8 step 2} X-Field <-> Data Pointer/HallSensorFieldsXYZ[{0..12 step 3}]  (5 links)
//     Term 21 (APS4322-7000)/Term 22 (APS4322-5000)/FB Inputs/A{0..8 step 2} Y-Field <-> Data Pointer/HallSensorFieldsXYZ[{1..13 step 3}]  (5 links)
//     Term 21 (APS4322-7000)/Term 22 (APS4322-5000)/FB Inputs/A{0..8 step 2} Z-Field <-> Data Pointer/HallSensorFieldsXYZ[{2..14 step 3}]  (5 links)
//     Term 21 (APS4322-7000)/Term 22 (APS4322-5000)/FB Inputs/B{1..9 step 2} X-Field <-> Data Pointer/HallSensorFieldsXYZ[{15..27 step 3}]  (5 links)
//     Term 21 (APS4322-7000)/Term 22 (APS4322-5000)/FB Inputs/B{1..9 step 2} Y-Field <-> Data Pointer/HallSensorFieldsXYZ[{16..28 step 3}]  (5 links)
//     Term 21 (APS4322-7000)/Term 22 (APS4322-5000)/FB Inputs/B{1..9 step 2} Z-Field <-> Data Pointer/HallSensorFieldsXYZ[{17..29 step 3}]  (5 links)
//     Term 21 (APS4322-7000)/Term 22 (APS4322-5000)/FB Inputs/C{0..8 step 2} X-Field <-> Data Pointer/HallSensorFieldsXYZ[{30..42 step 3}]  (5 links)
//     Term 21 (APS4322-7000)/Term 22 (APS4322-5000)/FB Inputs/C{0..8 step 2} Y-Field <-> Data Pointer/HallSensorFieldsXYZ[{31..43 step 3}]  (5 links)
//     Term 21 (APS4322-7000)/Term 22 (APS4322-5000)/FB Inputs/C{0..8 step 2} Z-Field <-> Data Pointer/HallSensorFieldsXYZ[{32..44 step 3}]  (5 links)
//     Term 21 (APS4322-7000)/Term 22 (APS4322-5000)/FB Inputs/D{1..9 step 2} X-Field <-> Data Pointer/HallSensorFieldsXYZ[{45..57 step 3}]  (5 links)
//     Term 21 (APS4322-7000)/Term 22 (APS4322-5000)/FB Inputs/D{1..9 step 2} Y-Field <-> Data Pointer/HallSensorFieldsXYZ[{46..58 step 3}]  (5 links)
//     Term 21 (APS4322-7000)/Term 22 (APS4322-5000)/FB Inputs/D{1..9 step 2} Z-Field <-> Data Pointer/HallSensorFieldsXYZ[{47..59 step 3}]  (5 links)
//     Term 21 (APS4322-7000)/Term 22 (APS4322-5000)/FB Inputs/E{0..8 step 2} X-Field <-> Data Pointer/HallSensorFieldsXYZ[{60..72 step 3}]  (5 links)
//     Term 21 (APS4322-7000)/Term 22 (APS4322-5000)/FB Inputs/E{0..8 step 2} Y-Field <-> Data Pointer/HallSensorFieldsXYZ[{61..73 step 3}]  (5 links)
//     Term 21 (APS4322-7000)/Term 22 (APS4322-5000)/FB Inputs/E{0..8 step 2} Z-Field <-> Data Pointer/HallSensorFieldsXYZ[{62..74 step 3}]  (5 links)
//     Term 21 (APS4322-7000)/Term 22 (APS4322-5000)/FB Inputs/F{1..9 step 2} X-Field <-> Data Pointer/HallSensorFieldsXYZ[{75..87 step 3}]  (5 links)
//     Term 21 (APS4322-7000)/Term 22 (APS4322-5000)/FB Inputs/F{1..9 step 2} Y-Field <-> Data Pointer/HallSensorFieldsXYZ[{76..88 step 3}]  (5 links)
//     Term 21 (APS4322-7000)/Term 22 (APS4322-5000)/FB Inputs/F{1..9 step 2} Z-Field <-> Data Pointer/HallSensorFieldsXYZ[{77..89 step 3}]  (5 links)
//     Term 21 (APS4322-7000)/Term 22 (APS4322-5000)/FB Inputs/G{0..8 step 2} X-Field <-> Data Pointer/HallSensorFieldsXYZ[{90..102 step 3}]  (5 links)
//     Term 21 (APS4322-7000)/Term 22 (APS4322-5000)/FB Inputs/G{0..8 step 2} Y-Field <-> Data Pointer/HallSensorFieldsXYZ[{91..103 step 3}]  (5 links)
//     Term 21 (APS4322-7000)/Term 22 (APS4322-5000)/FB Inputs/G{0..8 step 2} Z-Field <-> Data Pointer/HallSensorFieldsXYZ[{92..104 step 3}]  (5 links)
//     Term 21 (APS4322-7000)/Term 22 (APS4322-5000)/FB Inputs/H{1..9 step 2} X-Field <-> Data Pointer/HallSensorFieldsXYZ[{105..117 step 3}]  (5 links)
//     Term 21 (APS4322-7000)/Term 22 (APS4322-5000)/FB Inputs/H{1..9 step 2} Y-Field <-> Data Pointer/HallSensorFieldsXYZ[{106..118 step 3}]  (5 links)
//     Term 21 (APS4322-7000)/Term 22 (APS4322-5000)/FB Inputs/H{1..9 step 2} Z-Field <-> Data Pointer/HallSensorFieldsXYZ[{107..119 step 3}]  (5 links)
//     Term 21 (APS4322-7000)/Term 22 (APS4322-5000)/FB Inputs/I{0..8 step 2} X-Field <-> Data Pointer/HallSensorFieldsXYZ[{120..132 step 3}]  (5 links)
//     Term 21 (APS4322-7000)/Term 22 (APS4322-5000)/FB Inputs/I{0..8 step 2} Y-Field <-> Data Pointer/HallSensorFieldsXYZ[{121..133 step 3}]  (5 links)
//     Term 21 (APS4322-7000)/Term 22 (APS4322-5000)/FB Inputs/I{0..8 step 2} Z-Field <-> Data Pointer/HallSensorFieldsXYZ[{122..134 step 3}]  (5 links)
//     Term 21 (APS4322-7000)/Term 22 (APS4322-5000)/FB Inputs/J{1..9 step 2} X-Field <-> Data Pointer/HallSensorFieldsXYZ[{135..147 step 3}]  (5 links)
//     Term 21 (APS4322-7000)/Term 22 (APS4322-5000)/FB Inputs/J{1..9 step 2} Y-Field <-> Data Pointer/HallSensorFieldsXYZ[{136..148 step 3}]  (5 links)
//     Term 21 (APS4322-7000)/Term 22 (APS4322-5000)/FB Inputs/J{1..9 step 2} Z-Field <-> Data Pointer/HallSensorFieldsXYZ[{137..149 step 3}]  (5 links)
//     Term 21 (APS4322-7000)/Term 22 (APS4322-5000)/FB Inputs/Status <-> Data Pointer/FeedbackStatus
//   Device 2 (EtherCAT) <-> TcCOM Objects/XPlanar/Part1/Tile8
//     Term 23 (APS4322-7000)/APS Comm Inputs/CommStatusWord <-> Data Pointer/MoverCommStatusWord
//     Term 23 (APS4322-7000)/APS Comm Inputs/Data {1..4} <-> Data Pointer/MoverCommDataIn[{0..3}]  (4 links)
//     Term 23 (APS4322-7000)/APS Comm Outputs/CommControlWord <-> Data Pointer/MoverCommControlWord
//     Term 23 (APS4322-7000)/APS Comm Outputs/Data 1 <-> Data Pointer/MoverCommDataOut
//     Term 23 (APS4322-7000)/APS Diagdata/DC Link Voltage <-> Data Pointer/DcLinkVoltage
//     Term 23 (APS4322-7000)/APS Diagdata/Power supply current <-> Data Pointer/PowerSupplyCurrent
//     Term 23 (APS4322-7000)/APS Inputs/StatusWord <-> Data Pointer/PowerUnitStatusWord
//     Term 23 (APS4322-7000)/APS Outputs/ControlWord <-> Data Pointer/PowerUnitControlWord
//     Term 23 (APS4322-7000)/APS Outputs/Current D 0X0 <-> Data Pointer/DCurrentSetPoints[0]
//     Term 23 (APS4322-7000)/APS Outputs/Current D 0X1 <-> Data Pointer/DCurrentSetPoints[1]
//     Term 23 (APS4322-7000)/APS Outputs/Current D 0X2 <-> Data Pointer/DCurrentSetPoints[2]
//     Term 23 (APS4322-7000)/APS Outputs/Current D 1X0 <-> Data Pointer/DCurrentSetPoints[6]
//     Term 23 (APS4322-7000)/APS Outputs/Current D 1X1 <-> Data Pointer/DCurrentSetPoints[7]
//     Term 23 (APS4322-7000)/APS Outputs/Current D 1X2 <-> Data Pointer/DCurrentSetPoints[8]
//     Term 23 (APS4322-7000)/APS Outputs/Current D 2X0 <-> Data Pointer/DCurrentSetPoints[12]
//     Term 23 (APS4322-7000)/APS Outputs/Current D 2X1 <-> Data Pointer/DCurrentSetPoints[13]
//     Term 23 (APS4322-7000)/APS Outputs/Current D 2X2 <-> Data Pointer/DCurrentSetPoints[14]
//     Term 23 (APS4322-7000)/APS Outputs/Current D 3X0 <-> Data Pointer/DCurrentSetPoints[18]
//     Term 23 (APS4322-7000)/APS Outputs/Current D 3X1 <-> Data Pointer/DCurrentSetPoints[19]
//     Term 23 (APS4322-7000)/APS Outputs/Current D 3X2 <-> Data Pointer/DCurrentSetPoints[20]
//     Term 23 (APS4322-7000)/APS Outputs/Current D 0Y0 <-> Data Pointer/DCurrentSetPoints[3]
//     Term 23 (APS4322-7000)/APS Outputs/Current D 0Y1 <-> Data Pointer/DCurrentSetPoints[4]
//     Term 23 (APS4322-7000)/APS Outputs/Current D 0Y2 <-> Data Pointer/DCurrentSetPoints[5]
//     Term 23 (APS4322-7000)/APS Outputs/Current D 1Y0 <-> Data Pointer/DCurrentSetPoints[9]
//     Term 23 (APS4322-7000)/APS Outputs/Current D 1Y1 <-> Data Pointer/DCurrentSetPoints[10]
//     Term 23 (APS4322-7000)/APS Outputs/Current D 1Y2 <-> Data Pointer/DCurrentSetPoints[11]
//     Term 23 (APS4322-7000)/APS Outputs/Current D 2Y0 <-> Data Pointer/DCurrentSetPoints[15]
//     Term 23 (APS4322-7000)/APS Outputs/Current D 2Y1 <-> Data Pointer/DCurrentSetPoints[16]
//     Term 23 (APS4322-7000)/APS Outputs/Current D 2Y2 <-> Data Pointer/DCurrentSetPoints[17]
//     Term 23 (APS4322-7000)/APS Outputs/Current D 3Y0 <-> Data Pointer/DCurrentSetPoints[21]
//     Term 23 (APS4322-7000)/APS Outputs/Current D 3Y1 <-> Data Pointer/DCurrentSetPoints[22]
//     Term 23 (APS4322-7000)/APS Outputs/Current D 3Y2 <-> Data Pointer/DCurrentSetPoints[23]
//     Term 23 (APS4322-7000)/APS Outputs/Current Q 0X0 <-> Data Pointer/QCurrentSetPoints[0]
//     Term 23 (APS4322-7000)/APS Outputs/Current Q 0X1 <-> Data Pointer/QCurrentSetPoints[1]
//     Term 23 (APS4322-7000)/APS Outputs/Current Q 0X2 <-> Data Pointer/QCurrentSetPoints[2]
//     Term 23 (APS4322-7000)/APS Outputs/Current Q 1X0 <-> Data Pointer/QCurrentSetPoints[6]
//     Term 23 (APS4322-7000)/APS Outputs/Current Q 1X1 <-> Data Pointer/QCurrentSetPoints[7]
//     Term 23 (APS4322-7000)/APS Outputs/Current Q 1X2 <-> Data Pointer/QCurrentSetPoints[8]
//     Term 23 (APS4322-7000)/APS Outputs/Current Q 2X0 <-> Data Pointer/QCurrentSetPoints[12]
//     Term 23 (APS4322-7000)/APS Outputs/Current Q 2X1 <-> Data Pointer/QCurrentSetPoints[13]
//     Term 23 (APS4322-7000)/APS Outputs/Current Q 2X2 <-> Data Pointer/QCurrentSetPoints[14]
//     Term 23 (APS4322-7000)/APS Outputs/Current Q 3X0 <-> Data Pointer/QCurrentSetPoints[18]
//     Term 23 (APS4322-7000)/APS Outputs/Current Q 3X1 <-> Data Pointer/QCurrentSetPoints[19]
//     Term 23 (APS4322-7000)/APS Outputs/Current Q 3X2 <-> Data Pointer/QCurrentSetPoints[20]
//     Term 23 (APS4322-7000)/APS Outputs/Current Q 0Y0 <-> Data Pointer/QCurrentSetPoints[3]
//     Term 23 (APS4322-7000)/APS Outputs/Current Q 0Y1 <-> Data Pointer/QCurrentSetPoints[4]
//     Term 23 (APS4322-7000)/APS Outputs/Current Q 0Y2 <-> Data Pointer/QCurrentSetPoints[5]
//     Term 23 (APS4322-7000)/APS Outputs/Current Q 1Y0 <-> Data Pointer/QCurrentSetPoints[9]
//     Term 23 (APS4322-7000)/APS Outputs/Current Q 1Y1 <-> Data Pointer/QCurrentSetPoints[10]
//     Term 23 (APS4322-7000)/APS Outputs/Current Q 1Y2 <-> Data Pointer/QCurrentSetPoints[11]
//     Term 23 (APS4322-7000)/APS Outputs/Current Q 2Y0 <-> Data Pointer/QCurrentSetPoints[15]
//     Term 23 (APS4322-7000)/APS Outputs/Current Q 2Y1 <-> Data Pointer/QCurrentSetPoints[16]
//     Term 23 (APS4322-7000)/APS Outputs/Current Q 2Y2 <-> Data Pointer/QCurrentSetPoints[17]
//     Term 23 (APS4322-7000)/APS Outputs/Current Q 3Y0 <-> Data Pointer/QCurrentSetPoints[21]
//     Term 23 (APS4322-7000)/APS Outputs/Current Q 3Y1 <-> Data Pointer/QCurrentSetPoints[22]
//     Term 23 (APS4322-7000)/APS Outputs/Current Q 3Y2 <-> Data Pointer/QCurrentSetPoints[23]
//     Term 23 (APS4322-7000)/APS Outputs/PhiE 0X0 <-> Data Pointer/PhiSetPoints[0]
//     Term 23 (APS4322-7000)/APS Outputs/PhiE 0X1 <-> Data Pointer/PhiSetPoints[1]
//     Term 23 (APS4322-7000)/APS Outputs/PhiE 0X2 <-> Data Pointer/PhiSetPoints[2]
//     Term 23 (APS4322-7000)/APS Outputs/PhiE 1X0 <-> Data Pointer/PhiSetPoints[6]
//     Term 23 (APS4322-7000)/APS Outputs/PhiE 1X1 <-> Data Pointer/PhiSetPoints[7]
//     Term 23 (APS4322-7000)/APS Outputs/PhiE 1X2 <-> Data Pointer/PhiSetPoints[8]
//     Term 23 (APS4322-7000)/APS Outputs/PhiE 2X0 <-> Data Pointer/PhiSetPoints[12]
//     Term 23 (APS4322-7000)/APS Outputs/PhiE 2X1 <-> Data Pointer/PhiSetPoints[13]
//     Term 23 (APS4322-7000)/APS Outputs/PhiE 2X2 <-> Data Pointer/PhiSetPoints[14]
//     Term 23 (APS4322-7000)/APS Outputs/PhiE 3X0 <-> Data Pointer/PhiSetPoints[18]
//     Term 23 (APS4322-7000)/APS Outputs/PhiE 3X1 <-> Data Pointer/PhiSetPoints[19]
//     Term 23 (APS4322-7000)/APS Outputs/PhiE 3X2 <-> Data Pointer/PhiSetPoints[20]
//     Term 23 (APS4322-7000)/APS Outputs/PhiE 0Y0 <-> Data Pointer/PhiSetPoints[3]
//     Term 23 (APS4322-7000)/APS Outputs/PhiE 0Y1 <-> Data Pointer/PhiSetPoints[4]
//     Term 23 (APS4322-7000)/APS Outputs/PhiE 0Y2 <-> Data Pointer/PhiSetPoints[5]
//     Term 23 (APS4322-7000)/APS Outputs/PhiE 1Y0 <-> Data Pointer/PhiSetPoints[9]
//     Term 23 (APS4322-7000)/APS Outputs/PhiE 1Y1 <-> Data Pointer/PhiSetPoints[10]
//     Term 23 (APS4322-7000)/APS Outputs/PhiE 1Y2 <-> Data Pointer/PhiSetPoints[11]
//     Term 23 (APS4322-7000)/APS Outputs/PhiE 2Y0 <-> Data Pointer/PhiSetPoints[15]
//     Term 23 (APS4322-7000)/APS Outputs/PhiE 2Y1 <-> Data Pointer/PhiSetPoints[16]
//     Term 23 (APS4322-7000)/APS Outputs/PhiE 2Y2 <-> Data Pointer/PhiSetPoints[17]
//     Term 23 (APS4322-7000)/APS Outputs/PhiE 3Y0 <-> Data Pointer/PhiSetPoints[21]
//     Term 23 (APS4322-7000)/APS Outputs/PhiE 3Y1 <-> Data Pointer/PhiSetPoints[22]
//     Term 23 (APS4322-7000)/APS Outputs/PhiE 3Y2 <-> Data Pointer/PhiSetPoints[23]
//     Term 23 (APS4322-7000)/Term 24 (APS4322-5000)/FB Inputs/A{0..8 step 2} X-Field <-> Data Pointer/HallSensorFieldsXYZ[{0..12 step 3}]  (5 links)
//     Term 23 (APS4322-7000)/Term 24 (APS4322-5000)/FB Inputs/A{0..8 step 2} Y-Field <-> Data Pointer/HallSensorFieldsXYZ[{1..13 step 3}]  (5 links)
//     Term 23 (APS4322-7000)/Term 24 (APS4322-5000)/FB Inputs/A{0..8 step 2} Z-Field <-> Data Pointer/HallSensorFieldsXYZ[{2..14 step 3}]  (5 links)
//     Term 23 (APS4322-7000)/Term 24 (APS4322-5000)/FB Inputs/B{1..9 step 2} X-Field <-> Data Pointer/HallSensorFieldsXYZ[{15..27 step 3}]  (5 links)
//     Term 23 (APS4322-7000)/Term 24 (APS4322-5000)/FB Inputs/B{1..9 step 2} Y-Field <-> Data Pointer/HallSensorFieldsXYZ[{16..28 step 3}]  (5 links)
//     Term 23 (APS4322-7000)/Term 24 (APS4322-5000)/FB Inputs/B{1..9 step 2} Z-Field <-> Data Pointer/HallSensorFieldsXYZ[{17..29 step 3}]  (5 links)
//     Term 23 (APS4322-7000)/Term 24 (APS4322-5000)/FB Inputs/C{0..8 step 2} X-Field <-> Data Pointer/HallSensorFieldsXYZ[{30..42 step 3}]  (5 links)
//     Term 23 (APS4322-7000)/Term 24 (APS4322-5000)/FB Inputs/C{0..8 step 2} Y-Field <-> Data Pointer/HallSensorFieldsXYZ[{31..43 step 3}]  (5 links)
//     Term 23 (APS4322-7000)/Term 24 (APS4322-5000)/FB Inputs/C{0..8 step 2} Z-Field <-> Data Pointer/HallSensorFieldsXYZ[{32..44 step 3}]  (5 links)
//     Term 23 (APS4322-7000)/Term 24 (APS4322-5000)/FB Inputs/D{1..9 step 2} X-Field <-> Data Pointer/HallSensorFieldsXYZ[{45..57 step 3}]  (5 links)
//     Term 23 (APS4322-7000)/Term 24 (APS4322-5000)/FB Inputs/D{1..9 step 2} Y-Field <-> Data Pointer/HallSensorFieldsXYZ[{46..58 step 3}]  (5 links)
//     Term 23 (APS4322-7000)/Term 24 (APS4322-5000)/FB Inputs/D{1..9 step 2} Z-Field <-> Data Pointer/HallSensorFieldsXYZ[{47..59 step 3}]  (5 links)
//     Term 23 (APS4322-7000)/Term 24 (APS4322-5000)/FB Inputs/E{0..8 step 2} X-Field <-> Data Pointer/HallSensorFieldsXYZ[{60..72 step 3}]  (5 links)
//     Term 23 (APS4322-7000)/Term 24 (APS4322-5000)/FB Inputs/E{0..8 step 2} Y-Field <-> Data Pointer/HallSensorFieldsXYZ[{61..73 step 3}]  (5 links)
//     Term 23 (APS4322-7000)/Term 24 (APS4322-5000)/FB Inputs/E{0..8 step 2} Z-Field <-> Data Pointer/HallSensorFieldsXYZ[{62..74 step 3}]  (5 links)
//     Term 23 (APS4322-7000)/Term 24 (APS4322-5000)/FB Inputs/F{1..9 step 2} X-Field <-> Data Pointer/HallSensorFieldsXYZ[{75..87 step 3}]  (5 links)
//     Term 23 (APS4322-7000)/Term 24 (APS4322-5000)/FB Inputs/F{1..9 step 2} Y-Field <-> Data Pointer/HallSensorFieldsXYZ[{76..88 step 3}]  (5 links)
//     Term 23 (APS4322-7000)/Term 24 (APS4322-5000)/FB Inputs/F{1..9 step 2} Z-Field <-> Data Pointer/HallSensorFieldsXYZ[{77..89 step 3}]  (5 links)
//     Term 23 (APS4322-7000)/Term 24 (APS4322-5000)/FB Inputs/G{0..8 step 2} X-Field <-> Data Pointer/HallSensorFieldsXYZ[{90..102 step 3}]  (5 links)
//     Term 23 (APS4322-7000)/Term 24 (APS4322-5000)/FB Inputs/G{0..8 step 2} Y-Field <-> Data Pointer/HallSensorFieldsXYZ[{91..103 step 3}]  (5 links)
//     Term 23 (APS4322-7000)/Term 24 (APS4322-5000)/FB Inputs/G{0..8 step 2} Z-Field <-> Data Pointer/HallSensorFieldsXYZ[{92..104 step 3}]  (5 links)
//     Term 23 (APS4322-7000)/Term 24 (APS4322-5000)/FB Inputs/H{1..9 step 2} X-Field <-> Data Pointer/HallSensorFieldsXYZ[{105..117 step 3}]  (5 links)
//     Term 23 (APS4322-7000)/Term 24 (APS4322-5000)/FB Inputs/H{1..9 step 2} Y-Field <-> Data Pointer/HallSensorFieldsXYZ[{106..118 step 3}]  (5 links)
//     Term 23 (APS4322-7000)/Term 24 (APS4322-5000)/FB Inputs/H{1..9 step 2} Z-Field <-> Data Pointer/HallSensorFieldsXYZ[{107..119 step 3}]  (5 links)
//     Term 23 (APS4322-7000)/Term 24 (APS4322-5000)/FB Inputs/I{0..8 step 2} X-Field <-> Data Pointer/HallSensorFieldsXYZ[{120..132 step 3}]  (5 links)
//     Term 23 (APS4322-7000)/Term 24 (APS4322-5000)/FB Inputs/I{0..8 step 2} Y-Field <-> Data Pointer/HallSensorFieldsXYZ[{121..133 step 3}]  (5 links)
//     Term 23 (APS4322-7000)/Term 24 (APS4322-5000)/FB Inputs/I{0..8 step 2} Z-Field <-> Data Pointer/HallSensorFieldsXYZ[{122..134 step 3}]  (5 links)
//     Term 23 (APS4322-7000)/Term 24 (APS4322-5000)/FB Inputs/J{1..9 step 2} X-Field <-> Data Pointer/HallSensorFieldsXYZ[{135..147 step 3}]  (5 links)
//     Term 23 (APS4322-7000)/Term 24 (APS4322-5000)/FB Inputs/J{1..9 step 2} Y-Field <-> Data Pointer/HallSensorFieldsXYZ[{136..148 step 3}]  (5 links)
//     Term 23 (APS4322-7000)/Term 24 (APS4322-5000)/FB Inputs/J{1..9 step 2} Z-Field <-> Data Pointer/HallSensorFieldsXYZ[{137..149 step 3}]  (5 links)
//     Term 23 (APS4322-7000)/Term 24 (APS4322-5000)/FB Inputs/Status <-> Data Pointer/FeedbackStatus
//   XPlanar MC Project/Axes/Mover4330_1 <-> TcCOM Objects/XPlanar/Mover4330_1
//     IoToMc/STD <-> OutputsToNC3/HWToNC3
//   XPlanar MC Project/Axes/Mover4330_2 <-> TcCOM Objects/XPlanar/Mover4330_2
//     McToIo/STD <-> InputsFromNC3/NC3ToHW
//   XPlanar MC Project/Axes/Mover4330_3 <-> TcCOM Objects/XPlanar/Mover4330_3
//     IoToMc/STD <-> OutputsToNC3/HWToNC3
//     McToIo/STD <-> InputsFromNC3/NC3ToHW
//   XPlanar MC Project/Axes/Mover4330_4 <-> TcCOM Objects/XPlanar/Mover4330_4
//     McToIo/STD <-> InputsFromNC3/NC3ToHW
//   SMXPlanarMoverTest/SMXPlanarMoverTest Instance <-> Device 1 (EtherCAT)/Term 1 (EK1200)/Term 2 (EL9222-9482)
//     PlcTask Inputs/MAIN.EL9222_9482.MDP5001_922_Input/MDP5001_922_OCP_Inputs_Channel_1_Status <-> OCP Inputs Channel 2/Status
//   SMXPlanarMoverTest/SMXPlanarMoverTest Instance <-> Device 1 (EtherCAT)/Term 1 (EK1200)/Term 3 (EL9222-6600)
//     PlcTask Inputs/MAIN.EL9222_6600.MDP5001_922_Input/MDP5001_922_OCP_Inputs_Channel_1_Status <-> OCP Inputs Channel 2/Status
//   SMXPlanarMoverTest/SMXPlanarMoverTest Instance <-> XPlanar MC Project/Axes/Mover4330_1
//     PlcTask Inputs/MAIN.fbApp.fbMover1.MCTOPLC/ACT <-> McToPlc/ACT
//     PlcTask Inputs/MAIN.fbApp.fbMover1.MCTOPLC/COORDMODE <-> McToPlc/COORDMODE
//     PlcTask Inputs/MAIN.fbApp.fbMover1.MCTOPLC/SET <-> McToPlc/SET
//     PlcTask Inputs/MAIN.fbApp.fbMover1.MCTOPLC/SETONTRACK <-> McToPlc/SETONTRACK
//     PlcTask Inputs/MAIN.fbApp.fbMover1.MCTOPLC/STD <-> McToPlc/STD
//     PlcTask Outputs/MAIN.fbApp.fbMover1.PLCTOMC/STD <-> PlcToMc/STD
//   SMXPlanarMoverTest/SMXPlanarMoverTest Instance <-> XPlanar MC Project/Axes/Mover4330_2
//     PlcTask Inputs/MAIN.fbApp.fbMover2.MCTOPLC/ACT <-> McToPlc/ACT
//     PlcTask Inputs/MAIN.fbApp.fbMover2.MCTOPLC/COORDMODE <-> McToPlc/COORDMODE
//     PlcTask Inputs/MAIN.fbApp.fbMover2.MCTOPLC/SET <-> McToPlc/SET
//     PlcTask Inputs/MAIN.fbApp.fbMover2.MCTOPLC/SETONTRACK <-> McToPlc/SETONTRACK
//     PlcTask Inputs/MAIN.fbApp.fbMover2.MCTOPLC/STD <-> McToPlc/STD
//     PlcTask Outputs/MAIN.fbApp.fbMover2.PLCTOMC/STD <-> PlcToMc/STD
//   SMXPlanarMoverTest/SMXPlanarMoverTest Instance <-> XPlanar MC Project/Axes/Mover4330_3
//     PlcTask Inputs/MAIN.fbApp.fbMover3.MCTOPLC/ACT <-> McToPlc/ACT
//     PlcTask Inputs/MAIN.fbApp.fbMover3.MCTOPLC/COORDMODE <-> McToPlc/COORDMODE
//     PlcTask Inputs/MAIN.fbApp.fbMover3.MCTOPLC/SET <-> McToPlc/SET
//     PlcTask Inputs/MAIN.fbApp.fbMover3.MCTOPLC/SETONTRACK <-> McToPlc/SETONTRACK
//     PlcTask Inputs/MAIN.fbApp.fbMover3.MCTOPLC/STD <-> McToPlc/STD
//     PlcTask Outputs/MAIN.fbApp.fbMover3.PLCTOMC/STD <-> PlcToMc/STD
//   SMXPlanarMoverTest/SMXPlanarMoverTest Instance <-> XPlanar MC Project/Axes/Mover4330_4
//     PlcTask Inputs/MAIN.fbApp.fbMover4.MCTOPLC/ACT <-> McToPlc/ACT
//     PlcTask Inputs/MAIN.fbApp.fbMover4.MCTOPLC/COORDMODE <-> McToPlc/COORDMODE
//     PlcTask Inputs/MAIN.fbApp.fbMover4.MCTOPLC/SET <-> McToPlc/SET
//     PlcTask Inputs/MAIN.fbApp.fbMover4.MCTOPLC/SETONTRACK <-> McToPlc/SETONTRACK
//     PlcTask Inputs/MAIN.fbApp.fbMover4.MCTOPLC/STD <-> McToPlc/STD
//     PlcTask Outputs/MAIN.fbApp.fbMover4.PLCTOMC/STD <-> PlcToMc/STD
//   SMXPlanarMoverTest/SMXPlanarMoverTest Instance <-> XPlanar MC Project/Groups/Environment
//     PlcTask Inputs/MAIN.fbApp.fbEnvironment.MCTOPLC_STD <-> McToPlc/STD
//   SMXPlanarMoverTest/SMXPlanarMoverTest Instance <-> XPlanar MC Project/Groups/XPlanar
//     PlcTask Inputs/MAIN.fbApp.fbGroup.MCTOPLC_STD <-> McToPlc/STD
//   TcCOM Objects/XPlanar/Mover4330_1 <-> XPlanar MC Project/Axes/Mover4330_1
//     InputsFromNC3/NC3ToHW <-> McToIo/STD
//   TcCOM Objects/XPlanar/Mover4330_2 <-> XPlanar MC Project/Axes/Mover4330_2
//     OutputsToNC3/HWToNC3 <-> IoToMc/STD
//   TcCOM Objects/XPlanar/Mover4330_4 <-> XPlanar MC Project/Axes/Mover4330_4
//     OutputsToNC3/HWToNC3 <-> IoToMc/STD

CONFIGURATION SMXPlanarMoverTest
    RESOURCE PLC ON TwinCAT3
        TASK PlcTask(INTERVAL := T#10ms, PRIORITY := 21);
        PROGRAM MAIN WITH PlcTask : MAIN;
    END_RESOURCE
END_CONFIGURATION

// ---- DUTs/SpaceMouseInputs.TcDUT
TYPE SpaceMouseInputs :
STRUCT
	X	: INT;
	Y	: INT;
	Z	: INT;
	A	: INT;
	B	: INT;
	C	: INT;
	Btn1	: BOOL;
	Btn2	: BOOL;
END_STRUCT
END_TYPE

// ---- GVLs/GVL_XPlanarConstants.TcGVL

VAR_GLOBAL CONSTANT
	
	TileWidth : INT :=240;
	TileHeight	: INT := 240;
	MaxXYVelocity	: LREAL := 100.0;
	MaxZABCVelocity	: LREAL	:= 10.0;
	MaxAccerlation	: LREAL := 100.0;
	delta	: LREAL := 0.01;
	zPosMax	: LREAL := 4;
	zPosMin : LREAL := 0;
	fAngleAB	: LREAL :=0;
END_VAR

// ---- POUs/MAIN.TcPOU
PROGRAM MAIN
VAR
	stMouseInputs	: SpaceMouseInputs;
	fbApp	: XplanarJoystickInput;
	bInit	: BOOL;
	EL9222_9482	: MDP5001_922_D0074435;
	EL9222_6600	: MDP5001_922_D0074435;
END_VAR

IF NOT bInit THEN
	fbApp.MouseInputs REF= stMouseInputs;
	bInit := TRUE;
END_IF

IF bInit THEN
fbApp.Cycle();
END_IF

END_PROGRAM

// ---- POUs/XplanarJoystickInput.TcPOU
FUNCTION_BLOCK XplanarJoystickInput

VAR	
	_stMouseInputs	: REFERENCE TO SpaceMouseInputs;
	fbMover1	: MC_PlanarMover;
	fbMover2	: MC_PlanarMover;
	fbMover3	: MC_PlanarMover;
	fbMover4	: MC_PlanarMover;
	nState		: INT;
	slogMsg1	: STRING;
	slogMsg2	: STRING;
	slogMsg3	: STRING;
	slogMsg4	: STRING;
	fbFeedback1	: MC_PlanarFeedback;
	fbEnvFeedback	: MC_PlanarFeedback;
	fbGrpFeedback	: MC_PlanarFeedback;
	stOptions1	: ST_ExternalSetpointGenerationOptions;
	stPos2		: PositionXYC;
	stPos3		: PositionXYC;
	stPos4		: PositionXYC;
	
	stPosSnap1	: MoverVector;
	bMouseInput	: BOOL;
	fbEnvironment: MC_PlanarEnvironment;
	fbGroup		: MC_PlanarGroup;
	
END_VAR

METHOD AddStators : BOOL
VAR_INPUT
	X	: INT;
	Y	: INT;
END_VAR
VAR
	TileWidth	: INT := 240;
	TileHeight	: INT :=240;
	xCount		: INT;
	yCount		: INT;
END_VAR
FOR yCount := 0 TO Y-1 DO
	FOR xCount := 0 TO X-1 DO
fbEnvironment.AddStator(fbEnvFeedback, TileWidth*xCount,TileHeight*yCount);
	END_FOR
END_FOR
fbEnvironment.CreateBoundary(fbEnvFeedback);
END_METHOD

METHOD Cycle : BOOL
VAR_INPUT
END_VAR
CASE nState OF
	5:
		fbGroup.Enable(fbGrpFeedback);
		nState := 6;
	6:
		fbGrpFeedback.Update();
		IF fbGrpFeedback.Done THEN
		nState := 10;
		ELSIF fbGrpFeedback.Error THEN
			nState :=15;
		END_IF
	10:
		IF fbGroup.MCTOPLC_STD.GroupObjectCount = 0 THEN
		addStators(4,3);
		fbEnvironment.AddToGroup(fbEnvFeedback, fbGroup);
		END_IF
		
		
		
		stOptions1.mode := MC_SET_POSITION_MODE.Absolute;
		fbMover1.Enable(fbFeedback1);
		nState := 11;
	
	11:
		fbFeedback1.Update();
		IF fbFeedback1.Done THEN
			IF fbGroup.MCTOPLC_STD.GroupObjectCount = 1 THEN
			fbMover1.AddToGroup(fbFeedback1,fbGroup);
			END_IF
			nState := 12;
		ELSIF fbFeedback1.Error THEN
			nState := 15;
		END_IF
	12:
		fbFeedback1.Update();
		IF fbFeedback1.Done THEN
			nState := 20;
		ELSIF fbFeedback1.Error THEN
			nState := 15;
		END_IF
	20:
		SpaceMouseInput();
		//nState := 21; 

	IF _stMouseInputs.Btn2 THEN
		nState := 40;
	END_IF
	
	(*
	30:
		stPos1.SetValuesXYC(240,120,0);
		fbMover1.MoveToPosition(slogmsg1,stpos1,200,1000,1000,10000);
		nState := 31;
	31:
		IF fbMover1.P_MoveToPosition.Done THEN
			nState := 20;
		ELSIF fbMover1.P_MoveToPosition.Error THEN
			nState := 15;
		END_IF
	*)
	40:
		
		snapRotations();
		IF NOT bMouseInput THEN
			nState := 20;
		END_IF
	41:
		IF fbfeedBack1.Done THEN
			_stMouseInputs.Btn2 := FALSE;	
			nState := 20;
		ELSIF fbFeedback1.Error THEN
			_stMouseInputs.Btn2 := FALSE;
			nState := 15;
		END_IF
		
	42:
		fbMover1.Reset(fbFeedBack1);
		fbGroup.Reset(fbGrpFeedback);
		nState := 5;
		
END_CASE
fbGrpFeedback.Update();
fbEnvFeedback.Update();
fbFeedback1.Update();
fbEnvironment.Update();
fbGroup.Update();
fbMover1.Update();
END_METHOD

PROPERTY MouseInputs : REFERENCE TO SpaceMouseInputs
SET
IF __ISVALIDREF(MouseInputs) THEN
_stMouseInputs REF= MouseInputs;
END_IF
END_SET
END_PROPERTY

METHOD ScaleInput : LREAL
VAR_INPUT
	Input	: INT;
	ScaleRange		: LREAL;
END_VAR
VAR
	ScaleMax		: LREAL		:= 350;
END_VAR
scaleInput := INT_TO_LREAL(Input)*(ScaleRange/ScaleMax);
END_METHOD

METHOD SetAcceleration : BOOL;
VAR_INPUT
	Acceleration	: REFERENCE TO MoverVector;
	ZPos	: REFERENCE TO LREAL;
END_VAR
Acceleration.x := 0;
Acceleration.y := 0;
Acceleration.z := 0;
Acceleration.a := 0;
Acceleration.b := 0;
Acceleration.c := 0;
IF _stMouseInputs.X <-20 OR _stMouseInputs.X >20 THEN
	Acceleration.x := 100;
END_IF
IF _stMouseInputs.Y <-20 OR _stMouseInputs.Y >20 THEN
Acceleration.y := 100;
END_IF
IF (_stMouseInputs.Z <-20 AND ZPos > 0) OR (_stMouseInputs.Z >20 AND ZPos <4) THEN
Acceleration.z := 100;
END_IF
IF _stMouseInputs.A <-20 OR _stMouseInputs.A >20 THEN
Acceleration.a := 100;
END_IF
IF _stMouseInputs.B <-20 OR _stMouseInputs.B >20 THEN
Acceleration.b := 100;
END_IF
IF _stMouseInputs.C <-20 OR _stMouseInputs.C >20 THEN
Acceleration.c := 100;
END_IF
END_METHOD

METHOD SetPosition : BOOL
VAR_INPUT
	Position	: REFERENCE TO MoverVector;
END_VAR
VAR
	deltap		: LREAL := 0.008;
	deltan		: LREAL	:= -0.008;	
END_VAR
Position := fbMover1.MCTOPLC.ACT.ActPos;


IF _stMouseInputs.X > 20 THEN
	Position.x := Position.x + delta * scaleInput(ABS(_stMouseInputs.X),MaxXYVelocity);
ELSIF _stMouseInputs.X < -20 THEN
	Position.x := Position.x + (-1*delta * scaleInput(ABS(_stMouseInputs.X),MaxXYVelocity));
END_IF

IF _stMouseInputs.Y > 20 THEN
	Position.y := Position.y + delta * scaleInput(ABS(_stMouseInputs.Y),MaxXYVelocity);
ELSIF _stMouseInputs.Y < -20 THEN
	Position.y := Position.y + (-1*delta * scaleInput(ABS(_stMouseInputs.Y),MaxXYVelocity));
END_IF

IF _stMouseInputs.Z > 20 AND Position.z < 4 THEN
	Position.z := Position.z + delta * scaleInput(ABS(_stMouseInputs.Z),MaxZABCVelocity);
ELSIF _stMouseInputs.Z < -20 AND Position.z > 0 THEN
	Position.z := Position.z + (-1 * delta * scaleInput(ABS(_stMouseInputs.Z),MaxZABCVelocity));
END_IF

IF _stMouseInputs.A > 20 THEN
	Position.a := Position.a + delta * scaleInput(ABS(_stMouseInputs.A),MaxZABCVelocity);
ELSIF _stMouseInputs.A < -20 THEN
	Position.a := Position.a + (-1* delta * scaleInput(ABS(_stMouseInputs.A),MaxZABCVelocity));
END_IF

IF _stMouseInputs.B > 20 THEN
	Position.b := Position.b + delta * scaleInput(ABS(_stMouseInputs.B),MaxZABCVelocity);
ELSIF _stMouseInputs.B < -20 THEN
	Position.b := Position.b + (-1* delta * scaleInput(ABS(_stMouseInputs.B),MaxZABCVelocity));
END_IF

IF _stMouseInputs.C > 20 THEN
	Position.c := Position.c + delta * scaleInput(ABS(_stMouseInputs.C),MaxZABCVelocity);
ELSIF _stMouseInputs.C < -20 THEN
	Position.c := Position.c + (-1* delta * scaleInput(ABS(_stMouseInputs.C),MaxZABCVelocity));
END_IF
END_METHOD

METHOD SetVelocity : BOOL
VAR_INPUT
	Velocity	: REFERENCE TO MoverVector;
	ZPos		: REFERENCE TO LREAL;
END_VAR
VAR
		lTScale		: LREAL := 100.0;
		RScale		: LREAL := 10.0;
END_VAR
Velocity.x := 0;
Velocity.y := 0;
Velocity.z := 0;
Velocity.a := 0;
Velocity.b := 0;
Velocity.c := 0;

IF _stMouseInputs.X > 20 THEN
	Velocity.x := scaleInput(ABS(_stMouseInputs.X), MaxXYVelocity);
ELSIF _stMouseInputs.X < -20 THEN
	Velocity.x := ( -1 *scaleInput(ABS(_stMouseInputs.X), MaxXYVelocity));
END_IF

IF _stMouseInputs.Y > 20 AND ZPos < 4 THEN
	Velocity.y := scaleInput(ABS(_stMouseInputs.Y), MaxXYVelocity);
ELSIF _stMouseInputs.Y < -20 AND ZPos > 0 THEN
	Velocity.y := (-1 * scaleInput(ABS(_stMouseInputs.Y), MaxXYVelocity));
END_IF

IF _stMouseInputs.Z > 20 THEN
	Velocity.z := scaleInput(ABS(_stMouseInputs.Z), MaxZABCVelocity);
ELSIF _stMouseInputs.Z < -20 THEN
	Velocity.z := (-1 * scaleInput(ABS(_stMouseInputs.Z), MaxZABCVelocity));
END_IF

IF  _stMouseInputs.A > 20 THEN
	Velocity.a := scaleInput(ABS(_stMouseInputs.A), MaxZABCVelocity);
ELSIF _stMouseInputs.A < -20 THEN
	Velocity.a := (-1 *scaleInput(ABS(_stMouseInputs.A), MaxZABCVelocity));
END_IF

IF _stMouseInputs.B > 20THEN
	Velocity.b := scaleInput(ABS(_stMouseInputs.B), MaxZABCVelocity);
ELSIF  _stMouseInputs.B < -20  THEN
	Velocity.b := (-1 *scaleInput(ABS(_stMouseInputs.B), MaxZABCVelocity));
END_IF

IF _stMouseInputs.C > 20THEN
	Velocity.c := scaleInput(ABS(_stMouseInputs.C), MaxZABCVelocity);
ELSIF _stMouseInputs.C < -20 THEN
	Velocity.c := (-1 * scaleInput(ABS(_stMouseInputs.C), MaxZABCVelocity));
END_IF
END_METHOD

METHOD SnapRotations : BOOL
VAR
	
	Position	: MoverVector;
	Velocity	: MoverVector;
	Acceleration	: MoverVector;
	lMargin	: LREAL := 0.1;
	bADone	: BOOL;
	bBDone	: BOOL;
	bCDone	: BOOL;
	
END_VAR
VAR_INST
	fAngleC	:	LREAL;
END_VAR
stPosSnap1 := fbMover1.MCTOPLC.ACT.ActPos;

Velocity.x := 0;
Velocity.y := 0;
Velocity.z := 0;
Velocity.a := 0;
Velocity.b := 0;		
Velocity.c := 0;

Acceleration.x := 0;
Acceleration.y := 0;
Acceleration.z := 0;
Acceleration.a := 0;
Acceleration.b := 0;
Acceleration.c := 0;	
//IF stPosSnap1.c < -1.0 OR stPosSnap1.c > 1.0 THEN
//First cycle since snap command.

	IF _stMouseInputs.Btn2 AND NOT bMouseInput THEN
		fAngleC := snapTo90(stPosSnap1.c);
		fbMover1.StartExternalSetpointGeneration(fbFeedback1,stOptions1);
		bMouseInput := TRUE;
	END_IF
//make sure the difference between the nearest 90 degree angle and the curent position is great enough to command the mover to rotate.
IF (stPosSnap1.a >=0 AND stPosSnap1.a < fAngleAB + lMargin) OR (stPosSnap1.a <0 AND stPosSnap1.a > fAngleAB - lMargin) THEN
			bADone := TRUE;
END_IF
IF (stPosSnap1.b >=0 AND stPosSnap1.b < fAngleAB + lMargin) OR (stPosSnap1.b <0 AND stPosSnap1.b > fAngleAB - lMargin) THEN
			bBDone := TRUE;
END_IF
IF (stPosSnap1.c >=0 AND stPosSnap1.c < fAngleC + lMargin) OR (stPosSnap1.c <0 AND stPosSnap1.c > fAngleC - lMargin) THEN
		bCDone := TRUE;
END_IF
IF bADone AND bBDone AND bCDone THEN
	_stMouseInputs.Btn2 := FALSE;
END_IF

//Last cycle to end snap command
	IF NOT _stMouseInputs.Btn2 AND bMouseInput THEN
		Position := stPosSnap1;
		//Position.c := fAngleC;
		Velocity.a := 0;
		Velocity.b := 0;
		Velocity.c := 0;
		Acceleration.a := 0;
		Acceleration.b := 0;
		Acceleration.c := 0;
		fbMover1.SetExternalSetpoint(Position,Velocity,Acceleration);
		fbMover1.StopExternalSetpointGeneration(fbFeedback1);
		bMouseInput := FALSE;
	
	
	END_IF

	IF _stMouseInputs.Btn2 AND bMouseInput THEN
		
		Position := stPosSnap1;
		IF NOT bCDone THEN
			Acceleration.c := 100;
			IF (stPosSnap1.c - fAngleC) > 0 THEN
				Velocity.c := MaxZABCVelocity *-1;
			ELSIF (stPosSnap1.c - fAngleC) < 0 THEN
				Velocity.c := MaxZABCVelocity;
			END_IF
			
			IF stPosSnap1.c < 0 THEN
				Position.c := stPosSnap1.c + ((stPosSnap1.c - fAngleC) * ((-1*delta) * Velocity.c));
			ELSIF stPosSnap1.c > 0 THEN
				Position.c := stPosSnap1.c + ((stPosSnap1.c - fAngleC) * (delta * Velocity.c));
			END_IF
		END_IF
		
		IF NOT bADone THEN 
			Acceleration.a := 100;
			IF (stPosSnap1.a - fAngleAB) > 0 THEN
				Velocity.a := MaxZABCVelocity *-1;
			ELSIF (stPosSnap1.a - fAngleAB) < 0 THEN
				Velocity.a := MaxZABCVelocity;
			END_IF
			IF stPosSnap1.a < 0 THEN
			Position.a := stPosSnap1.a + ((stPosSnap1.a - fAngleAB) * ((-1*delta) * Velocity.a));
		ELSIF stPosSnap1.a > 0 THEN
			Position.a := stPosSnap1.a + ((stPosSnap1.a - fAngleAB) * (delta * Velocity.a));
		END_IF
		END_IF
		
		IF NOT bBDone THEN
			Acceleration.b := 100;
			IF (stPosSnap1.b - fAngleAB) > 0 THEN
				Velocity.b := MaxZABCVelocity *-1;
			ELSIF (stPosSnap1.b - fAngleAB) < 0 THEN
				Velocity.b := MaxZABCVelocity;
			END_IF
			IF stPosSnap1.b < 0 THEN
				Position.b := stPosSnap1.b + ((stPosSnap1.b - fAngleAB) * ((-1*delta) * Velocity.b));
			ELSIF stPosSnap1.b > 0 THEN
				Position.b := stPosSnap1.b + ((stPosSnap1.b - fAngleAB) * (delta * Velocity.b));
			END_IF
	
		END_IF
		
		fbMover1.SetExternalSetpoint(Position,Velocity,Acceleration);
	END_IF
END_METHOD

METHOD SnapTo90 : LREAL
VAR_INPUT
	fInput : LREAL;
END_VAR
VAR
	fResult	: LREAL;
	nTurns	: DINT;
	fRemainder	: LREAL;
	fTurnAngle	: LREAL := 90.0;
END_VAR
nTurns := MODTURNS(fInput,fTurnAngle);
fRemainder := LMOD(fInput,fTurnAngle);  
IF (nTurns > 0 AND fRemainder >= (fTurnAngle/2)) OR (nTurns <0 AND fRemainder >= (-1 * fTurnAngle/2))  THEN
	nTurns := nTurns + 1;
END_IF
fResult := nTurns * fTurnAngle;
snapTo90 := fResult;
END_METHOD

METHOD SpaceMouseInput : BOOL
VAR_INPUT
END_VAR
VAR 
	Position	: MoverVector;
	Velocity	: MoverVector;	
	Acceleration	: MoverVector;

END_VAR
IF 	_stMouseInputs.X < -20 OR _stMouseInputs.X > 20 OR
	_stMouseInputs.Y < -20 OR _stMouseInputs.Y > 20 OR
	_stMouseInputs.Z < -20 OR _stMouseInputs.Z > 20 OR 
	_stMouseInputs.A < -20 OR _stMouseInputs.A > 20 OR 
	_stMouseInputs.B < -20 OR _stMouseInputs.B > 20 OR 
	_stMouseInputs.C < -20 OR _stMouseInputs.C > 20 THEN
	
	IF NOT bMouseInput THEN
	
		fbMover1.StartExternalSetpointGeneration(fbFeedback1,stOptions1);
		bMouseInput := TRUE;
		Position := fbMover1.MCTOPLC.ACT.ActPos; Velocity.x := 0.0; Acceleration.x := 0.0;
		fbMover1.SetExternalSetpoint(Position,Velocity,Acceleration);
	ELSE	
		setPosition(Position);
		setVelocity(Velocity,Position.z);
		setAcceleration(Acceleration,Position.z);
		fbMover1.SetExternalSetpoint(Position,Velocity,Acceleration);
		
	END_IF
	
	
ELSE
	IF bMouseInput THEN	
		setPosition(Position);
		setVelocity(Velocity,Position.z);
		setAcceleration(Acceleration, Position.z);
		fbMover1.SetExternalSetpoint(Position,Velocity,Acceleration);
		fbMover1.StopExternalSetpointGeneration(fbFeedback1);
		bMouseInput := FALSE;
	END_IF
END_IF
END_METHOD

END_FUNCTION_BLOCK
